FUNCTION_BLOCK FB_CommandChangeStart EXTENDS FB_CommandChange IMPLEMENTS ITF_CommandChange
VAR

END_VAR

(*			
	RafalOS
	Rafał Osajda		03.11.2025		TC 4024.66
	Test czy można zmienić stan lub tryb i zwraca czy można i uruchamia zmianę
*)
METHOD PUBLIC Execute : BOOL
VAR_INPUT
	iNumberOfCommand	: INT;
END_VAR
IF (THIS^.itfSaMController.GetState () = E_BaseMachineState.Idle) THEN		// sprawdzenie czy jesteśmy w dobrym stanie dla tego rozkazu
	IF (THIS^.itfSaMController.IsStateInModeEnabled (eStateIn := E_BaseMachineState.Starting)) THEN	//test czy stan do którego chcemy przejśc jest właczony dla tego trybu
		THIS^.itfSaMController.ChangeStateTo (eStateIn := E_BaseMachineState.Starting);
	ELSE
		THIS^.EventSetActive (iNumber := 5);	//stan docelowy jest wylaczony w tym trybie
	END_IF
ELSE
	THIS^.EventSetActive (iNumber := 4);	//ten rozkaz nie obsluguje tego stanu
END_IF
END_METHOD

METHOD FB_init : BOOL
VAR_INPUT
	bInitRetains : BOOL; // if TRUE, the retain variables are initialized (warm start / cold start)
	bInCopyCode : BOOL;  // if TRUE, the instance afterwards gets moved into the copy code (online change)
END_VAR
THIS^.SetText (eLocation := E_BaseLocation.pl, wsDescription := "Command change state - Start");
THIS^.SetText (eLocation := E_BaseLocation.en, wsDescription := "Command change state - Start");
THIS^.SetText (eLocation := E_BaseLocation.de, wsDescription := "Command change state - Start");
THIS^.SetName (stName := THIS^.GetTexts ());
END_METHOD

END_FUNCTION_BLOCK

(* stored: Version 1.1.0.1
   POU FB_CommandChangeStart: Id {3e97eb6b-0aae-0d44-3f5a-d06acc717999}, SpecialFunc None
   Method Execute: Id {110a2e8c-d603-09b5-38f5-48392df7be8a}
   Method FB_init: Id {8a8b6ee8-32b2-028a-07da-958bf1cc3ceb} *)
